TEXTLIST KPickType
  0 = 'Pack'
  1 = 'Pallet'
  2 = 'Layer'
   = ''
END_TEXTLIST

(* stored: Version 1.1.0.1, ProductVersion 3.1.4024.11
   TextList KPickType: Id {61f76e91-1894-4353-bd19-1a5348c53297} *)
